Staubli VAL3: Emergencia.pgx

program Emergencia()
begin

  do
    if diAlarmaPlc==true

      taskKill("Principal")
      taskKill("N1_Home")
      taskKill("N10_AproBanyera")
      taskKill("N11_Banyera")
      taskKill("N12_AproAmpolla")
      taskKill("N13_Ampolla")
      taskKill("N15_AproAgafarPuntes")
      taskKill("N16_AgafarPuntes")
      taskKill("N17_AproTirarPuntes")
      taskKill("N18_TirarPuntes")
      taskKill("N20_AproDosi")
      taskKill("N21_Dosi")
      taskKill("N22_PosDosi")


      resetMotion()
      //Reset variables
      doRobotHome=false
      doRobotEnMoviment=false

      doAlarmaColisioRobot=false
      doTaskDone=false

      bTaskDone=false
      bPrimerCicle=false
      nSeqHome=0
      aioSet(aoProgramaRobot,0)
      aioSet(aoZonaHome,0)

      wait(diAlarmaPlc==false)

      taskCreate "Principal",50,Principal()
    endIf
    delay(0)
  until false


end
